FUNCTION_BLOCK PVDERATOR_PROP (* Proportional controller for PV power deration *)
  (* Standard: 61499-2 *)
  (* Version 0.0, 2017-06-15, Marc Jakobi, HTW Berlin *)
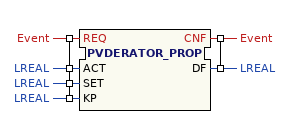
  EVENT_INPUT
    REQ WITH ACT, SET, KP; (* Normal Execution Request *)
  END_EVENT
  EVENT_OUTPUT
    CNF WITH DF; (* Execution Confirmation *)
  END_EVENT
  VAR_INPUT
    ACT : LREAL; (* Actual PV (feed-in) power in kW/kWp *)
    SET : LREAL; (* Set PV (feed-in) power in kW/kWp *)
    KP : LREAL; (* Proportional control coefficient *)
  END_VAR
  VAR_OUTPUT
    DF : LREAL := 1; (* Derating factor *)
  END_VAR
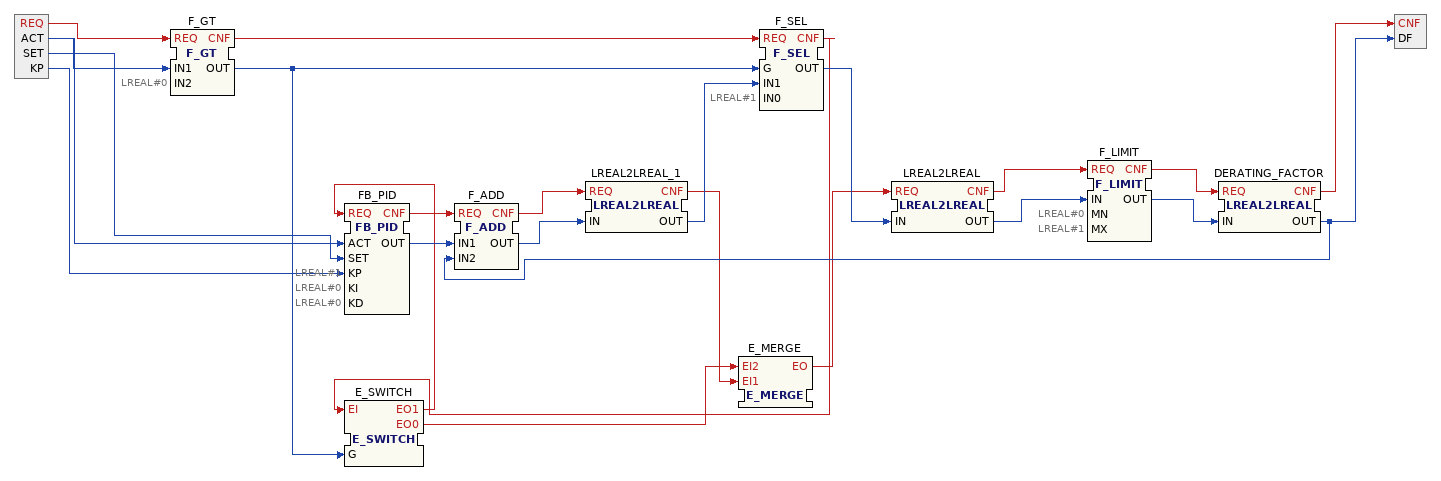
  FBS
    FB_PID : FB_PID(KP := LREAL#1, KI := LREAL#0, KD := LREAL#0);
    F_ADD : F_ADD;
    DERATING_FACTOR : LREAL2LREAL;
    F_LIMIT : F_LIMIT(MN := LREAL#0, MX := LREAL#1);
    LREAL2LREAL : LREAL2LREAL;
    F_GT : F_GT(IN2 := LREAL#0);
    F_SEL : F_SEL(IN0 := LREAL#1);
    E_SWITCH : E_SWITCH;
    LREAL2LREAL_1 : LREAL2LREAL;
    E_MERGE : E_MERGE;
  END_FBS
  EVENT_CONNECTIONS
    DERATING_FACTOR.CNF TO CNF;
    FB_PID.CNF TO F_ADD.REQ;
    REQ TO F_GT.REQ;
    F_GT.CNF TO F_SEL.REQ;
    F_SEL.CNF TO E_SWITCH.EI;
    E_SWITCH.EO1 TO FB_PID.REQ;
    E_SWITCH.EO0 TO E_MERGE.EI2;
    LREAL2LREAL_1.CNF TO E_MERGE.EI1;
    F_ADD.CNF TO LREAL2LREAL_1.REQ;
    E_MERGE.EO TO LREAL2LREAL.REQ;
    LREAL2LREAL.CNF TO F_LIMIT.REQ;
    F_LIMIT.CNF TO DERATING_FACTOR.REQ;
  END_CONNECTIONS
  DATA_CONNECTIONS
    ACT TO FB_PID.ACT;
    SET TO FB_PID.SET;
    DERATING_FACTOR.OUT TO DF;
    FB_PID.OUT TO F_ADD.IN1;
    ACT TO F_GT.IN1;
    F_GT.OUT TO F_SEL.G;
    DERATING_FACTOR.OUT TO F_ADD.IN2;
    F_GT.OUT TO E_SWITCH.G;
    LREAL2LREAL_1.OUT TO F_SEL.IN1;
    F_ADD.OUT TO LREAL2LREAL_1.IN;
    F_SEL.OUT TO LREAL2LREAL.IN;
    LREAL2LREAL.OUT TO F_LIMIT.IN;
    F_LIMIT.OUT TO DERATING_FACTOR.IN;
    KP TO FB_PID.KP;
  END_CONNECTIONS
END_FUNCTION_BLOCK
